KUKA KRL program: LAB_MINIMAL.src, LAB_MINIMAL.dat

--- LAB_MINIMAL.src ---
&ACCESS RVP
&REL 1
&PARAM TEMPLATE = C:\KRC\Roboter\Template\vorgabe
&PARAM EDITMASK = *
DEF LAB_MINIMAL()
  ; KLAB fixture: synthetic virtual-only PTP + LIN seed
  BAS(#INITMOV,0)
  $ADVANCE=3
  $IPO_MODE=#BASE
  $ORI_TYPE=#VAR
  BAS(#TOOL,0)
  BAS(#BASE,0)
  $ACC.CP=1.0
  $VEL.ORI1=100
  $VEL.ORI2=100
  $ACC.ORI1=100
  $ACC.ORI2=100
  $APO.CDIS=0
  $APO.CPTP=0
  BAS(#VEL_PTP,100)
  BAS(#ACC_PTP,100)
  ; Neutral BCO target: preserve the controller's current axis position.
  PTP $AXIS_ACT
  PTP A_HOME
  PTP P_START
  $VEL.CP=0.5
  LIN P_END
END

--- LAB_MINIMAL.dat ---
&ACCESS RVP
&REL 1
DEFDAT LAB_MINIMAL PUBLIC
  DECL E6AXIS A_HOME={A1 0,A2 -90,A3 90,A4 0,A5 0,A6 0,E1 0,E2 0,E3 0,E4 0,E5 0,E6 0}
  DECL E6POS P_START={X 1900,Y -100,Z 1200,A 180,B 0,C 180,S 2,T 2,E1 0,E2 0,E3 0,E4 0,E5 0,E6 0}
  DECL E6POS P_END={X 1900,Y 100,Z 1200,A 180,B 0,C 180,S 2,T 2,E1 0,E2 0,E3 0,E4 0,E5 0,E6 0}
ENDDAT
